PROGRAM DeviceState
VAR
	nDev1_DevState AT %I* : UINT;
	nDev4_DevState AT %I* : UINT;
	nProfinetState AT %I* : UINT;
	nPnIoBoxState AT %I* : UINT;
	nPnIoBoxCtrl AT %Q* : UINT;
	nState		: UINT;
	bReset		: BOOL;
	bErrorBit	: BOOL;
	tDelay		: TON;
	tPulse		: TON;
END_VAR

;
(*
bErrorBit		:= nPnIoBoxState.3;
nPnIoBoxCtrl.0	:= bReset;

CASE nState OF
	
	0:
	IF nProfinetState <> 8 OR bErrorBit THEN
		tDelay(IN:=TRUE , PT:=T#5S);
		IF tDelay.Q THEN
			tPulse(IN:=TRUE , PT:=T#1S);
			bReset	:= TRUE;
			nState	:= 10;
		END_IF
	ELSE
		tDelay(IN:=FALSE);	
	END_IF
	
	10:
	tPulse();
	IF tPulse.Q THEN
		bReset	:= FALSE;
		tDelay(IN:=FALSE);
		tPulse(IN:=FALSE);
		nState	:= 0;	
	END_IF
	
END_CASE
*)

END_PROGRAM

(* stored: Version 1.1.0.1, ProductVersion 3.1.4024.12
   POU DeviceState: Id {1859fefa-b38d-4207-adce-aabf25f3f954}, SpecialFunc None *)
